{attribute 'qualified_only'}
VAR_GLOBAL
	bInvisibleLockOpened:										BOOL;
	bInvisibleLockClosed:										BOOL;
	bInvisibleLockClosedAndQuit:								BOOL;
END_VAR

(* stored: Version 1.1.0.1, ProductVersion 3.1.4024.12
   GVL GVL_SAFETY: Id {3a335149-8470-4e9a-a532-9661bdecab34} *)
